//Fills an array of LREAL of varible length with zeros
FUNCTION ZEROS_INT
VAR_IN_OUT
	arr: ARRAY [*] OF INT;
END_VAR
VAR
	i : DINT := 0;
END_VAR

FOR i := LOWER_BOUND(arr,1) TO UPPER_BOUND(arr, 1) BY 1 DO
	arr[i] := 0;
END_FOR

END_FUNCTION

(* stored: Version 1.1.0.1, ProductVersion 3.1.4024.11
   POU ZEROS_INT: Id {ae10d378-96fe-4ac7-be99-5c473769a6eb}, SpecialFunc None *)
